{attribute 'GeneratedUsingTerminal: EK1100-0000-0018'}
{attribute addProperty BoxType "EK1100-0000-0018"}
{attribute addProperty Id "RC10_B1_EL7041_1000EL7041_86DE63E743RC10_B2_EL7041_1000EL7041_86DE63E743RC10_C11_EL7041_1000EL7041_86DE63E743RC10_C12_EL7041_1000EL7041_86DE63E743RC10_C21_EL7041_1000EL7041_86DE63E743RC10_C22_EL7041_1000EL7041_86DE63E743RC10_2_EndTerminal_EL9010EL9010_D29C20850"}
{attribute addProperty CRC "663114785"}
{attribute addProperty Size "258"}
{attribute addProperty Name "RC10_2 (EK1100)"}
TYPE RC10_2_EK1100_27865421 EXTENDS EK1100_1FC0878B :
STRUCT
	{attribute addProperty Name "RC10_B1 (EL7041-1000)"}
	{attribute addProperty PreviousPort "RC10_2 (EK1100) : B"}
	{attribute addProperty SyncUnit "C10"}
	RC10_B1_EL7041_1000 : EL7041_86DE63E7;
	{attribute addProperty Name "RC10_B2 (EL7041-1000)"}
	{attribute addProperty PreviousPort "RC10_B1 (EL7041-1000) : B"}
	{attribute addProperty SyncUnit "C10"}
	RC10_B2_EL7041_1000 : EL7041_86DE63E7;
	{attribute addProperty Name "RC10_C11 (EL7041-1000)"}
	{attribute addProperty PreviousPort "RC10_B2 (EL7041-1000) : B"}
	{attribute addProperty SyncUnit "C10"}
	RC10_C11_EL7041_1000 : EL7041_86DE63E7;
	{attribute addProperty Name "RC10_C12 (EL7041-1000)"}
	{attribute addProperty PreviousPort "RC10_C11 (EL7041-1000) : B"}
	{attribute addProperty SyncUnit "C10"}
	RC10_C12_EL7041_1000 : EL7041_86DE63E7;
	{attribute addProperty Name "RC10_C21 (EL7041-1000)"}
	{attribute addProperty PreviousPort "RC10_C12 (EL7041-1000) : B"}
	{attribute addProperty SyncUnit "C10"}
	RC10_C21_EL7041_1000 : EL7041_86DE63E7;
	{attribute addProperty Name "RC10_C22 (EL7041-1000)"}
	{attribute addProperty PreviousPort "RC10_C21 (EL7041-1000) : B"}
	{attribute addProperty SyncUnit "C10"}
	RC10_C22_EL7041_1000 : EL7041_86DE63E7;
	{attribute addProperty Name "RC10_2_EndTerminal (EL9010)"}
	{attribute addProperty PreviousPort "RC10_C22 (EL7041-1000) : B"}
	{attribute addProperty SyncUnit "default"}
	RC10_2_EndTerminal_EL9010 : EL9010_D29C2085;
END_STRUCT
END_TYPE

(* stored: Version 1.2.0.0, ProductVersion 3.1.4024.11
   DUT RC10_2_EK1100_27865421: Id {fc24514a-7aec-059e-39c1-edf5fbe38e41} *)
